FUNCTION_BLOCK FB_SameSizeCVCamera EXTENDS FB_ActionBasic
VAR_INPUT
    xExecute    : BOOL;
    xAbort      : BOOL;
	xReset		: BOOL;
    Cylinder 	: REFERENCE TO UNI_CylinderList;
    TimeOut  	: LREAL := 600; // Unit : s
	Input		: ST_InputTable;
	OutPut		: ST_OutputTable;
	Motor		: REFERENCE to UNI_MotorList;
	BoxCameraDone :BOOL;
END_VAR	
VAR_OUTPUT
    xAborted : BOOL;
    iErrorID : INT;
    ErrorMsg : STRING;
	UseBoxCamera	:BOOL;
END_VAR
VAR
    StateBehaviour   : CBML.ETrigATo;
    CurrentPosition : ST_PositionTable;
	uiCyclicStep    : UINT := 0;
	TON_DelaySensor	:TON;
	TON_TimeOut		:TON;
	TON_ArriviedTimeOut :TON ;
	TON_CameraTimeOut	:TON;
	TON_ConveyorTimeOut	:TON;
	Reset_Rtrig 	:R_TRIG;
	TON_SameSizeBoxDetect1_Delay :TON;
	fbExecuteEdgeDetect :FB_EdgeDetect;
	// ========== Resume 續做機制 ==========
	uiResumeStep	: UINT := 0;		// 錯誤發生時記錄的步驟，供續做使用
	bResumeEnabled	: BOOL := FALSE;	// 續做模式啟用旗標
END_VAR

THIS^.IBehaviourModel := StateBehaviour;

StateBehaviour(xExecute := xExecute,
              xAbort := xAbort OR fbExecuteEdgeDetect.xFallingEdge,
              udiTimeOut := LREAL_TO_UDINT( TimeOut*1000000),
              xDone => xDone,
              xBusy => xBusy,
              xError => xError,
              xAborted => xAborted);

fbExecuteEdgeDetect(xInput :=xExecute);

iErrorID := StateBehaviour._model.iErrorID;
ErrorMsg := M_GetErrorMsg(xErrorID := iErrorID);

Reset_Rtrig(CLK:= xReset);
IF Reset_Rtrig.Q THEN
	StateBehaviour.ResetModel(xCommit:=xReset);
END_IF

A00_BaseUnits();

ACTION A00_BaseUnits:
TON_DelaySensor(PT:= T#1S);
TON_TimeOut(PT := T#20S);
TON_ArriviedTimeOut(PT:= T#60S);
TON_CameraTimeOut(PT:=T#600S);
TON_ConveyorTimeOut(PT:=T#60S);
TON_SameSizeBoxDetect1_Delay(PT:=T#3S);
TON_SameSizeBoxDetect1_Delay.IN :=Input.bSameSizeCV_BoxDetect1_Sensor AND Motor.List.TransmitSameSideCV.InForWard;
END_ACTION

METHOD CleanupAction
VAR_INPUT
    xAbortProposed : BOOL;
    iErrorIDProposed: INT;
END_VAR
VAR_OUTPUT
    xComplete : BOOL := TRUE;
    xAbort: BOOL := xAbortProposed;
 	iErrorID : INT := iErrorIDProposed;
END_VAR
xComplete := FALSE;

// ============================================================
// Resume 機制：保存當前步驟供後續 Resume 使用
// ============================================================
IF uiResumeStep = 0 THEN
	uiResumeStep := uiCyclicStep;
END_IF

// 清除所有 Timer
TON_DelaySensor.IN 		:= FALSE;
TON_TimeOut.IN 			:= FALSE;
TON_ArriviedTimeOut.IN 	:= FALSE;
TON_CameraTimeOut.IN 	:= FALSE;
TON_ConveyorTimeOut.IN 	:= FALSE;

// 重置輸出信號
UseBoxCamera 	:= FALSE;
BoxCameraDone 	:= FALSE;

// 機械復位到安全狀態
Cylinder.List.fbSameSizeCV_Block1.M_Retract();
Cylinder.List.fbSameSizeCV_Block2.M_Retract();
Cylinder.List.fbSameSizeCV_Press1.M_Retract();
//Cylinder.List.fbSameSizeCV_Press2.M_Retract();
Cylinder.List.fbTransmitCV_CamaraHoriz.M_Retract();
Motor.List.TransmitSameSideCV.M_MotorStop();

// 等待機械復位完成
IF Cylinder.List.fbSameSizeCV_Block1.InRearPosition AND
   Cylinder.List.fbSameSizeCV_Block2.InRearPosition AND
   Cylinder.List.fbSameSizeCV_Press1.InRearPosition AND
   //Cylinder.List.fbSameSizeCV_Press2.InRearPosition AND
   Cylinder.List.fbTransmitCV_CamaraHoriz.InRearPosition AND
   Motor.List.TransmitSameSideCV.InStopped THEN
	xComplete := TRUE;
END_IF
END_METHOD

METHOD CyclicAction
VAR_INPUT
    itfTimingController : CBML.ITimingController;
END_VAR
VAR_OUTPUT
    xComplete : BOOL := TRUE;
    iErrorID : INT := 0;
END_VAR
VAR_INST
	bMoveConveyorForward:BOOL;
END_VAR
xComplete := FALSE;
IF bMoveConveyorForward THEN
	IF NOT Motor.List.TransmitSameSideCV.InBackWard THEN
		Motor.List.TransmitSameSideCV.M_MoveForward();
	END_IF
END_IF

CASE uiCyclicStep OF
	0:	// 初始化
		bMoveConveyorForward:=FALSE;
		uiCyclicStep :=1000;
		
	1000:	// 擋第一個盒子
		TON_TimeOut.IN:=TRUE;
		Cylinder.List.fbSameSizeCV_Block1.M_Extend();
		Cylinder.List.fbTransmitCV_CamaraHoriz.M_Retract();
		IF Cylinder.List.fbSameSizeCV_Block1.InFrontPosition AND
			Cylinder.List.fbTransmitCV_CamaraHoriz.InRearPosition THEN
			TON_TimeOut.IN:=FALSE;
			uiCyclicStep :=1050;
		END_IF
		IF TON_TimeOut.Q THEN
			uiResumeStep := uiCyclicStep;
			iErrorID := 7;
		END_IF

	1050:	// 馬達前進
		TON_ConveyorTimeOut.IN:=TRUE;
		bMoveConveyorForward:=TRUE;
		Cylinder.List.fbSameSizeCV_Press2.M_Retract();
		IF Motor.List.TransmitSameSideCV.InForWard AND
			Cylinder.List.fbSameSizeCV_Press2.InRearPosition THEN
			TON_ConveyorTimeOut.IN:= FALSE;
			uiCyclicStep :=1100;
		END_IF
		IF TON_ConveyorTimeOut.Q THEN
			uiResumeStep := uiCyclicStep;
			iErrorID := 7;
		END_IF

	1100:	// 檢查盒子到達擋塊
		TON_ArriviedTimeOut.IN:=TRUE;
		TON_DelaySensor.IN:=Input.bSameSizeCV_BoxDetect2_Sensor;
		IF TON_DelaySensor.Q THEN
			TON_DelaySensor.IN :=FALSE;
			TON_ArriviedTimeOut.IN :=FALSE;
			Cylinder.List.fbSameSizeCV_Press2.M_Extend();
			bMoveConveyorForward:=FALSE;
			Motor.List.TransmitSameSideCV.M_MotorStop();
			uiCyclicStep :=1200;
		END_IF
		IF TON_ArriviedTimeOut.Q THEN
			uiResumeStep := uiCyclicStep;
			iErrorID := 8;
		END_IF

	1200:	// 發送拍照請求 & 擋住第二個盒子
		TON_ConveyorTimeOut.IN:=TRUE;
		IF Cylinder.List.fbSameSizeCV_Press2.InFrontPosition AND
			Motor.List.TransmitSameSideCV.InStopped THEN
			TON_ConveyorTimeOut.IN:= FALSE;
			UseBoxCamera :=TRUE;
			uiCyclicStep :=1300;
		END_IF
		IF TON_ConveyorTimeOut.Q THEN
			uiResumeStep := uiCyclicStep;
			iErrorID := 9;
		END_IF

	1300:	// 等待 C# 拍照完成 (Camera 錯誤不可續做)
		TON_CameraTimeOut.IN:=TRUE;
		IF BoxCameraDone THEN
			TON_CameraTimeOut.IN :=FALSE;
			Cylinder.List.fbSameSizeCV_Block1.M_Retract();
			bMoveConveyorForward:=TRUE;
			uiCyclicStep :=1400;
		END_IF
		IF TON_CameraTimeOut.Q THEN
			uiResumeStep := uiCyclicStep;
			iErrorID :=10;
		END_IF

	1400:	// 盒子通過 Detect1 感測器
		TON_TimeOut.IN :=TRUE;
		IF Input.bSameSizeCV_BoxDetect1_Sensor THEN
			TON_TimeOut.IN :=FALSE;
			uiCyclicStep :=1500;
		END_IF
		IF TON_TimeOut.Q THEN
			uiResumeStep := uiCyclicStep;
			iErrorID :=11;
		END_IF

	1500:	// 離開感測器後停止馬達
		TON_DelaySensor.IN :=TRUE;
		IF NOT Input.bSameSizeCV_BoxDetect1_Sensor THEN
			TON_DelaySensor.IN :=FALSE;
			bMoveConveyorForward:=FALSE;
			Motor.List.TransmitSameSideCV.M_MotorStop();
			uiCyclicStep :=1600;
		END_IF
		IF TON_DelaySensor.Q THEN 
			TON_DelaySensor.IN:=FALSE;
			bMoveConveyorForward:=FALSE;
			Motor.List.TransmitSameSideCV.M_MotorStop();
			uiCyclicStep :=1600;
		END_IF
	
	1600:	// 等待馬達停止
		IF Motor.List.TransmitSameSideCV.InStopped THEN
			xComplete :=TRUE;
		END_IF

END_CASE

IF TON_SameSizeBoxDetect1_Delay.Q THEN
	iErrorID := 20;
END_IF
END_METHOD

METHOD ExitAction
VAR_INPUT
    xAfterCleanup : BOOL;
    xInCopyCode : BOOL;
END_VAR
	uiCyclicStep    := 0;
	xAfterCleanup := true;
END_METHOD

METHOD M_GetErrorMsg : T_MaxString
VAR_INPUT
	xErrorID: INT;
END_VAR

VAR
	
END_VAR
CASE xErrorID OF
	0:
		M_GetErrorMsg := 'No Error';
	1:
		M_GetErrorMsg := 'Action time out';
	2:
		M_GetErrorMsg := 'Position Data invalid';
	3:
		M_GetErrorMsg := 'Block1 cylinder not ready';
	4:
		M_GetErrorMsg := 'Block2 cylinder not ready';
	5:
		M_GetErrorMsg := 'Press1 cylinder not ready';
	6:
		M_GetErrorMsg := 'Press2 cylinder not ready';
	7:
		M_GetErrorMsg := 'CameraHoriz cylinder not ready';
	8:
		M_GetErrorMsg :='Conveyor not ready';
	9:
		M_GetErrorMsg :='Cylinder timeout';
	10:
		M_GetErrorMsg :='box not arrived timeout';
	11:
		M_GetErrorMsg :='Cylinder timeout';
	12:
		M_GetErrorMsg :='C# send BoxCameraDone timeout';
	
		
	20:
		M_GetErrorMsg :='SameSizeConveyor full box infront ';
END_CASE
END_METHOD

METHOD ResetAction
VAR_OUTPUT
    xComplete : BOOL := TRUE;
END_VAR
xComplete := FALSE;

// ============================================================
// Resume 機制判斷
// ------------------------------------------------------------
// 當錯誤發生後，操作員可選擇：
//   1. 保持 xExecute = TRUE 並按 Reset → Resume (從錯誤點繼續)
//   2. 先關閉 xExecute，再重新啟動 → 從頭開始
// ============================================================
bResumeEnabled := xExecute;

// 如果不是 Resume 模式，清除 Resume 步驟記錄
IF NOT bResumeEnabled THEN
	uiResumeStep := 0;
END_IF

// 清除所有 Timer
TON_DelaySensor.IN 		:= FALSE;
TON_TimeOut.IN 			:= FALSE;
TON_ArriviedTimeOut.IN 	:= FALSE;
TON_CameraTimeOut.IN 	:= FALSE;
TON_ConveyorTimeOut.IN 	:= FALSE;

xComplete := TRUE;
END_METHOD

METHOD StartAction
VAR_OUTPUT
    xComplete : BOOL := TRUE;
	iErrorID : INT := 0;
END_VAR
VAR
	bIsResumeMode : BOOL;	// 局部變數：記錄是否為 Resume 模式
END_VAR
xComplete := FALSE;

// 清除所有 Timer
TON_DelaySensor.IN 		:= FALSE;
TON_TimeOut.IN 			:= FALSE;
TON_ArriviedTimeOut.IN 	:= FALSE;
TON_CameraTimeOut.IN 	:= FALSE;
TON_ConveyorTimeOut.IN 	:= FALSE;

// ============================================================
// Resume 機制處理
// ------------------------------------------------------------
// 可 Resume 的錯誤: Error 7, 8, 9, 11 (氣缸/馬達/等待盒子)
// 不可 Resume 的錯誤: Error 10 (C# 拍照失敗), Error 20 (輸送帶滿載)
// ============================================================
bIsResumeMode := bResumeEnabled AND uiResumeStep > 0 AND uiResumeStep <> 1300;

IF bResumeEnabled AND uiResumeStep > 0 THEN
	IF uiResumeStep = 1300 THEN
		// Camera 錯誤：不可 Resume，強制從頭開始
		uiCyclicStep 	:= 0;
		UseBoxCamera 	:= FALSE;
		BoxCameraDone 	:= FALSE;
	ELSE
		// 其他錯誤：允許 Resume (人工已確認可繼續)
		uiCyclicStep := uiResumeStep;
	END_IF
	// 清除 Resume 旗標
	bResumeEnabled 	:= FALSE;
	uiResumeStep 	:= 0;
ELSE
	// 正常模式：從頭開始
	uiCyclicStep 	:= 0;
	UseBoxCamera 	:= FALSE;
	BoxCameraDone 	:= FALSE;
END_IF

// ============================================================
// 啟動前錯誤檢查
// ============================================================
IF TON_SameSizeBoxDetect1_Delay.Q THEN
	iErrorID := 20;
END_IF

IF Cylinder.List.fbSameSizeCV_Block1.xError THEN
	iErrorID := 3;
END_IF
IF Cylinder.List.fbSameSizeCV_Block2.xError THEN
	iErrorID := 4;
END_IF
IF Cylinder.List.fbSameSizeCV_Press1.xError THEN
	iErrorID := 5;
END_IF
IF Cylinder.List.fbSameSizeCV_Press2.xError THEN
	iErrorID := 6;
END_IF
IF Cylinder.List.fbTransmitCV_CamaraHoriz.xError THEN
	iErrorID := 7;
END_IF
IF Motor.List.TransmitSameSideCV.xError THEN
	iErrorID := 8;
END_IF

// 完成條件：Resume 模式直接完成，正常模式需檢查初始位置
IF bIsResumeMode OR
   (Cylinder.List.fbSameSizeCV_Block1.InRearPosition AND
    Motor.List.TransmitSameSideCV.InStopped) THEN
	xComplete := TRUE;
END_IF
END_METHOD

END_FUNCTION_BLOCK

(* stored: Version 1.1.0.1, ProductVersion 3.1.4024.13
   POU FB_SameSizeCVCamera: Id {b7f0f090-2562-464a-a72f-754890f967dc}, SpecialFunc None
   Folder Action: Id {909e43ed-f32f-4583-a821-5a821c77a293}
   Action A00_BaseUnits: Id {9ca21b52-2b9f-4cbd-86fd-c07e780d2cc5}
   Method CleanupAction: Id {b2d8576e-0acf-41ea-a7ea-005e6167ae00}
   Method CyclicAction: Id {83b7b3e0-663c-4997-991a-1e5f51179e2f}
   Method ExitAction: Id {27d4f9f7-8ed3-49e3-872f-64623caca5f5}
   Method M_GetErrorMsg: Id {39c43e65-7f65-40b7-8290-b8d4c7038d11}
   Method ResetAction: Id {800e20c2-a4b8-4568-b782-f7995ece63c5}
   Method StartAction: Id {28b648fd-dfe0-4659-ac89-9339de507591} *)
